// Mitsubishi GX Developer project: 1   PLC: FX2N

PROGRAM MAIN
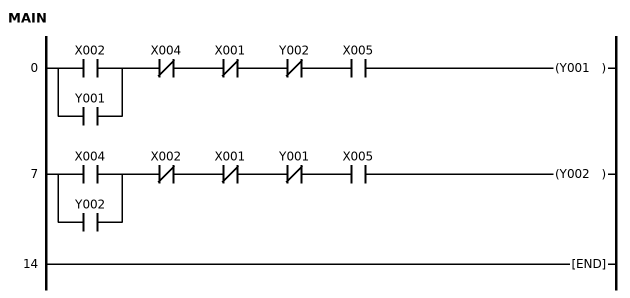
0     LD      X002
      OR      Y001
      ANI     X004
      ANI     X001
      ANI     Y002
      AND     X005
      OUT     Y001
7     LD      X004
      OR      Y002
      ANI     X002
      ANI     X001
      ANI     Y001
      AND     X005
      OUT     Y002
14    END
END_PROGRAM
